FUNCTION_BLOCK FB_Conveyor
VAR
	bRunning : BOOL := FALSE;
END_VAR

GVL_IO.bConveyorMotor := bRunning;

METHOD Start : BOOL
VAR_INPUT
END_VAR
bRunning := TRUE;
Start     := TRUE;
END_METHOD

METHOD Stop : BOOL
VAR_INPUT
END_VAR
bRunning := FALSE;
Stop      := TRUE;
END_METHOD

END_FUNCTION_BLOCK

(* stored: Version 1.1.0.1, ProductVersion 3.1.4024.16
   POU FB_Conveyor: Id {6e370f51-6d8d-403e-890f-ddf63c2f9544}, SpecialFunc None
   Method Start: Id {0046f898-0d7c-4f64-aa05-07ba9bceed5b}
   Method Stop: Id {b8dc2d25-3da3-4ee7-bda6-72b387173785} *)
